{attribute 'qualified_only'}
{attribute 'strict'}
TYPE CoreGripperControlState :
(
	Init,
	Open,
	Closing,
	Closed,
	Opening
);
END_TYPE

(* stored: Version 1.1.0.1, ProductVersion 3.1.4024.11
   DUT CoreGripperControlState: Id {818f4766-2336-4d30-8580-2ae2e5dc9048} *)
